FUNCTION_BLOCK fb_TimeStepUp
VAR_INPUT
	I_bExecute		:BOOL;
	I_nSteps		:LREAL := 0.1;
	I_nStart		:LREAL := 1;
	I_nMax			:LREAL := 4;
	I_tVerz			:TIME := T#10MS;
END_VAR
VAR_OUTPUT
	Q_nActStep		:LREAL;
END_VAR
VAR
	iStep	:INT;
	tonVerz	:ton;
END_VAR

tonVerz(
	PT := I_tVerz);

IF I_bExecute
THEN
	CASE iStep OF
	(*========================================*)
	0:	(* INIT *)	
		tonVerz.IN := FALSE;
		Q_nActStep := I_nStart;
		iStep := 1;
		
	(*========================================*)	
	1:	(* Step Up *)
		IF Q_nActStep < I_nMax
		THEN
			tonVerz.IN := TRUE;
			IF tonVerz.Q
			THEN
				Q_nActStep := Q_nActStep + I_nSteps;
				iStep := 2;
			END_IF
		ELSE
			Q_nActStep := I_nMax;
			iStep := 999;
		END_IF
		
	(*========================================*)	
	2:	(* ZURÜCK *)
		tonVerz.IN := FALSE;
		iStep := 1;
		
	(*========================================*)	
	999:(* ENDE *)	
		
	END_CASE
ELSE
	iStep := 0;
	Q_nActStep := I_nStart;
END_IF

END_FUNCTION_BLOCK

(* stored: Version 1.1.0.1, ProductVersion 3.1.4024.15
   POU fb_TimeStepUp: Id {4f1d5501-40be-4c09-ac6b-780c57586417}, SpecialFunc None *)
